FB_ReadXmlLineMsg(
	Prefix:= 'MSG',
	ID:= ,
	File:= 'MSG.xml',
	Text=>);

IF 	Error.Text<>'' THEN
	Error.Text:=CONCAT(Error.Text,sInit.InstName);
	Error.Text:=CONCAT(Error.Text,' :');
	Error.Text:=CONCAT(Error.Text,FB_ReadXmlLineConf.Text);
	Error.Text:=CONCAT(Error.Text,' - ');
	Error.Text:=CONCAT(Error.Text,FB_ReadXmlLineMsg.Text);
END_IF
END_FUNCTION_BLOCK

(* POU zLibrary/Sensopart/FB_Sensopart, ST *)
FUNCTION_BLOCK FB_Sensopart
VAR_INPUT
	b_init							: BOOL;
	b_start							: BOOL;
	b_start_manual					: BOOL;
	b_quitt							: BOOL;
	b_reset							: BOOL;
	b_kamera_aktiv 					: BOOL;
	i16_job							: INT:=1;
	st_Description					: STRING;
END_VAR
VAR_OUTPUT
	b_ready							: BOOL;
	b_done							: BOOL;
	b_busy							: BOOL;
	b_error							: BOOL;

(* Ausgänge der Kamera *)
	Ergebnis_IO						: BOOL;
	Ergebnis_NIO					: BOOL;
	sm_kamera_nicht_bb				: BOOL := FALSE;
	sm_zeitueberschreitung			: BOOL := FALSE;
END_VAR
VAR
	b_first_cycle					: BOOL := TRUE;
	fb_ton_quitt					: TON;
	fb_ton_trigger					: TON;
	fb_tof_trigger					: TOF;
	fb_state_entry					: ST_StateEntry;
	fb_r_trig_start					: R_TRIG;
	fb_r_trig_trigger				: R_TRIG;
END_VAR

VAR_OUTPUT
	(*Sensopart Kamera*)
	a_Trigger 				AT %Q*: BOOL;
	a_Job_Bit1 				AT %Q*: BOOL;
	a_Job_Bit2 				AT %Q*: BOOL;
	a_Job_Bit3 				AT %Q*: BOOL;
	a_Job_Bit4 				AT %Q*: BOOL;
END_VAR
VAR

(* Eingänge von der Kamera *)
	e_Ergebnis_iO			AT %I*: BOOL;
	e_Ergebnis_niO			AT %I*: BOOL;
	e_Betriebsbereit		AT %I*: BOOL;
	e_Best_Jobwechsel		AT %I*: BOOL;
END_VAR
IF b_first_cycle THEN
	b_first_cycle := FALSE;
END_IF

a_Job_Bit1:=i16_job.0;
a_Job_Bit2:=i16_job.1;
a_Job_Bit3:=i16_job.2;
a_Job_Bit4:=i16_job.3;

(* Zeiten *)
fb_ton_quitt(IN:= , PT:= t#100ms, Q=> , ET=> );
fb_ton_trigger(IN:= , PT:= t#150ms, Q=> , ET=> );
fb_tof_trigger(IN:= fb_r_trig_trigger.Q , PT:= t#150ms, Q=> , ET=> );

(* Flanken *)
fb_r_trig_start(CLK:= b_start OR b_start_manual, Q=> );


IF	NOT b_kamera_aktiv THEN
	fb_state_entry.i16_next_step := INAKTIV;
END_IF

(* ==================================Schrittkette================================ *)
fb_state_entry(i16_pos:= 1);

CASE fb_state_entry.i16_step OF
(*=======================================================*)
	INIT_OBJ:
		fb_state_entry.i16_next_step := INIT;

(*=======================================================*)
	INIT:
		IF 	fb_state_entry.E THEN
			b_ready := FALSE;
			b_done := FALSE;
			b_quitt := FALSE;
			b_reset := FALSE;
			b_busy := FALSE;
			b_error := FALSE;
			b_start := FALSE;
			a_Trigger  := FALSE;
			Ergebnis_IO := FALSE;
			Ergebnis_NIO := FALSE;
			sm_kamera_nicht_bb := FALSE;
			sm_zeitueberschreitung := FALSE;
		END_IF

		(*-----------------------Weiterschaltbedingungen----------------------------*)
		IF 	b_init THEN
			IF  NOT b_kamera_aktiv THEN
				fb_state_entry.i16_next_step := BEREIT;		(* Kamera ist inaktiv *)
			ELSE
				fb_state_entry.i16_next_step := 20;			(* Kamera ist aktiv *)
			END_IF
		END_IF

(*=======================================================*)
	20: fb_state_entry.s_debugtext:='Kurze Wartezeit';

		IF 	fb_state_entry.fb_ton_Step.ET > t#300ms THEN
			fb_state_entry.i16_next_step := 30;
		END_IF

(*=======================================================*)
	30: fb_state_entry.s_debugtext:='Kamera Betriebsbereit';

		(*-----------------------Weiterschaltbedingungen----------------------------*)
		IF 	e_Betriebsbereit THEN
			fb_state_entry.i16_next_step := BEREIT;
		ELSIF
		 	fb_state_entry.fb_ton_Step.ET > t#300ms THEN
			sm_kamera_nicht_bb := TRUE;
			fb_state_entry.i16_next_step := FEHLER;
		END_IF

(*=======================================================*)
	BEREIT: fb_state_entry.s_debugtext:='warte auf Start';

		IF fb_state_entry.E THEN
			b_ready := TRUE;
			b_done := TRUE;
		END_IF

		(*-----------------------Weiterschaltbedingungen----------------------------*)
		IF 	b_kamera_aktiv THEN			(* Kamera aktiv *)
			IF 	fb_r_trig_start.Q AND e_Betriebsbereit THEN
				b_start := FALSE;
				b_busy := TRUE;
				b_done := FALSE;
				Ergebnis_IO := FALSE;
				Ergebnis_NIO := FALSE;
				fb_state_entry.i16_next_step := 102;
			ELSIF
				NOT e_Betriebsbereit THEN
				sm_kamera_nicht_bb := TRUE;
				fb_state_entry.i16_next_step := FEHLER;
			END_IF
		ELSE							(* Simulation der Kamera *)
			IF 	fb_r_trig_start.Q THEN
				b_busy := TRUE;
				b_done := FALSE;
				b_start:=FALSE;
				Ergebnis_IO := FALSE;
				Ergebnis_NIO := FALSE;
				fb_state_entry.i16_next_step := 300;
			END_IF
		END_IF

(*=======================================================*)
	102: fb_state_entry.s_debugtext:='Jobwechsel';

		IF 	fb_state_entry.fb_ton_Step.ET > t#1s OR
			e_Best_Jobwechsel THEN
			fb_state_entry.i16_next_step := 105;
		END_IF

(*=======================================================*)
	105: fb_state_entry.s_debugtext:='Kamera wieder bereit';

		IF 	e_Betriebsbereit THEN
			fb_state_entry.i16_next_step := 110;
		ELSIF
			NOT e_Betriebsbereit AND fb_state_entry.fb_ton_Step.ET > t#2s THEN
			sm_kamera_nicht_bb := TRUE;
			fb_state_entry.i16_next_step := FEHLER;
		END_IF

(*=======================================================*)
	110: fb_state_entry.s_debugtext:='Trigger setzen ';

		IF 	fb_state_entry.E THEN
			a_Trigger := TRUE;
			Ergebnis_IO := FALSE;
			Ergebnis_NIO := FALSE;
			fb_ton_trigger.IN := TRUE;
		END_IF

		(*-----------------------Weiterschaltbedingungen----------------------------*)
		IF 	fb_ton_trigger.Q THEN
			a_Trigger := FALSE;
			fb_ton_trigger.IN := FALSE;
			fb_state_entry.i16_next_step := 130;
		END_IF

(*=======================================================*)
	120: fb_state_entry.s_debugtext:='Warten auf Ergebnis der Kamera';

		IF 	NOT e_Ergebnis_iO AND
			NOT e_Ergebnis_niO THEN
			fb_state_entry.i16_next_step := 130;
		ELSIF
			fb_state_entry.fb_ton_Step.ET > t#4000ms THEN
			sm_zeitueberschreitung := TRUE;
			fb_state_entry.i16_next_step := FEHLER;
		END_IF

(*=======================================================*)
	130: fb_state_entry.s_debugtext:='Warten auf Ergebnis der Kamera ';

		IF 	NOT fb_state_entry.E AND e_Ergebnis_iO AND e_Betriebsbereit THEN
			Ergebnis_IO := TRUE;
			fb_state_entry.i16_next_step := BEREIT;
		ELSIF
			NOT fb_state_entry.E AND e_Ergebnis_niO AND e_Betriebsbereit THEN
			Ergebnis_NIO := TRUE;
			fb_state_entry.i16_next_step := BEREIT;
		ELSIF
			fb_state_entry.fb_ton_Step.ET > t#4000ms THEN
			sm_zeitueberschreitung := TRUE;
			fb_state_entry.i16_next_step := FEHLER;
		END_IF

		IF 	fb_state_entry.X THEN
			b_busy := FALSE;
			b_done := TRUE;
		END_IF

(*=======================================================*)
	300: fb_state_entry.s_debugtext:='Kamera ist nicht aktiv (Warten) ';		

		IF 	fb_state_entry.fb_ton_Step.ET > t#500ms THEN
			b_busy := FALSE;
			b_done := TRUE;
			Ergebnis_IO := TRUE;
			fb_state_entry.i16_next_step := BEREIT;
		END_IF

(*=======================================================*)
	STOP, FEHLER:
		IF 	fb_state_entry.E THEN
			b_error := TRUE;
			fb_ton_quitt.IN := FALSE;
			a_Trigger := FALSE;
		END_IF

		(*-----------------------Weiterschaltbedingungen----------------------------*)
		IF	(b_reset OR b_quitt) AND
			NOT fb_state_entry.E THEN
			b_error := FALSE;
			fb_ton_quitt.IN := TRUE;
		END_IF

		IF 	fb_ton_quitt.Q THEN
			fb_ton_quitt.IN := FALSE;
			fb_state_entry.i16_next_step := INIT;
		END_IF

(*=======================================================*)
	INAKTIV:
		IF 	fb_state_entry.E THEN
			b_ready := FALSE;
			b_done := FALSE;
			b_busy := FALSE;
			b_start := FALSE;
		END_IF

		IF	b_kamera_aktiv THEN
			fb_state_entry.i16_next_step := STOP;
		END_IF

END_CASE

fb_state_entry(i16_pos:= 2);
END_FUNCTION_BLOCK

(* POU zLibrary/Sensopart/FB_SensopartEthernet, ST *)
FUNCTION_BLOCK FB_SensopartEthernet
VAR_INPUT
	Activated				: BOOL;
	JobNo					: INT;
	s_IpAdress				: STRING;
	i_DataPort				: UDINT;
	i_CmdPort				: UDINT;
	st_ctrl_in				: struct_ctrl_in;
	st_Description			: STRING;
	st_InstName				: STRING;
	SensopartErgebnis		: STRING(15); (*Ergebnis Sensopart Kamera*)
END_VAR
VAR_IN_OUT

END_VAR
VAR_OUTPUT
	st_ctrl_out				: struct_ctrl_out;
	Connected				: BOOL;							(* Sockets Connected*)
	RecvDataString			: T_MaxString;
	ActJobNo				: INT;
END_VAR
VAR
	fb_ton_quitt						: TON;
	fb_state_entry					: ST_StateEntry;
	fb_state_entry_command			: ST_StateEntry;

	(* Error Handling *)
	FB_ReadXmlLineConf			: FB_ReadXmlLine;
	FB_ReadXmlLineMsg			: FB_ReadXmlLine;
	(*Variablen für Behr Meldungen*)
	TempErrorText					: STRING(255);
	ProcessTime					: DINT;				(* Counts the time in steps of 100ms since starting operation *)
	Error							: ErrorStruct;

	sm_kamera_keine_reaktion		: BOOL;
	sm_kamera_nicht_bb			: BOOL;
	sm_jobnummer_nicht_erlaubt		: BOOL;		(* erlaubter Bereich von 1-255 *)
	sm_kamera_command_error		: BOOL;
	sm_kamera_connect_error		: BOOL;
	sm_kamera_send_error			: BOOL;
	sm_kamera_rec_error			: BOOL;

	(*TcpIp-Connection via Socket*)
	FBClientServerConnectionCmd 	: FB_ClientServerConnection;
	FBClientServerConnectionRcv 	: FB_ClientServerConnection;
	FBSocketSend					: FB_SocketSend;
	FBSocketRecv					: FB_SocketReceive;
	SocketHandleCmd				: T_HSOCKET;
	SocketHandleRcv				: T_HSOCKET;
	ErrorId						: UDINT;
	nRecBytes					: UDINT;						(* Contains the number of bytes currently received. *)

	RecvStringCmd				: STRING(25);

	TRG_CMD:		ARRAY [0..2] OF BYTE:= 16#54,16#52,16#47;	(* [T, R, G] Trigger *)
	CJB_CMD:		ARRAY [0..5] OF BYTE:= 16#43,16#4A,16#42;	(* [C, J, B, 0, 0, 1] ChangeJoB z.B für Jobnummer 1 *)
	CJB_RCV:		ARRAY [0..7] OF BYTE;

	JbNoMem					: INT;
	CalcJbNo					: BYTE;

	b_Kam_Pruef_IO			:BOOL; 				(* Kameraprüfung Ergebnis iO *)
	b_Kam_Pruef_NIO			:BOOL; 				(* Kameraprüfung Ergebnis niO *)

	b_Kam_Bereit	  			: BOOL;				(* Bereit für nächsten ext. Trigger *)
	b_Betriebsbereit_eth			: BOOL:=FALSE;	(* Bereit kommt von EtherNet (noch nicht programmiert) *)
	e_Betriebsbereit  		AT %I*: BOOL;			(* Bereit kommt nur über Hardware-Eingang *)
 	BtnConnect					: sButtonVisu;
	BtnTrigger					: sButtonVisu;

END_VAR
(* Zeiten *)
fb_ton_quitt(IN:= , PT:= t#100ms, Q=> , ET=> );

(* Aufrufe *)
Btn_Init();
Command();
ErrorHandling();

b_Kam_Bereit := e_Betriebsbereit OR b_Betriebsbereit_eth;	(* Betriebsbereit  von EtherNet oder Eingang *)

(* Toplevel *)
IF	NOT Activated THEN
	fb_state_entry.i16_next_step := INAKTIV;
END_IF

IF fb_state_entry.i16_next_step > INIT AND fb_state_entry.i16_next_step < FEHLER THEN
	IF fb_state_entry.i16_next_step < STOP THEN
		IF st_ctrl_in.b_stop THEN
			fb_state_entry.i16_next_step := STOP;
		END_IF
		IF 	sm_kamera_command_error OR
			sm_kamera_send_error OR
			sm_kamera_rec_error OR
			sm_kamera_connect_error THEN
			fb_state_entry.i16_next_step := FEHLER;
		END_IF
	END_IF
END_IF

(* ==================================Schrittkette================================ *)
fb_state_entry(i16_pos:= 1);

CASE fb_state_entry.i16_step OF
(*=======================================================*)
INIT_OBJ:

	fb_state_entry.i16_next_step := INIT;

(*=======================================================*)
INIT:
	IF 	fb_state_entry.E THEN
		fb_ton_quitt.IN := FALSE;
		st_ctrl_out := st_ctrl_out_Empty;
		b_Kam_Pruef_IO := FALSE;
		b_Kam_Pruef_NIO := FALSE;
		sm_kamera_nicht_bb := FALSE;
		sm_kamera_keine_reaktion := FALSE;
		sm_jobnummer_nicht_erlaubt := FALSE;
		sm_kamera_command_error:=FALSE;
		sm_kamera_connect_error:=FALSE;
		sm_kamera_send_error:=FALSE;
		sm_kamera_rec_error:=FALSE;
		Error.No:=0;
		Error.Text:='';
	END_IF

	(*-----------------------Weiterschaltbedingungen----------------------------*)
	IF	BtnConnect.tasten OR
		st_ctrl_in.b_init THEN
		fb_state_entry.i16_next_step := 30;
	END_IF

(*=======================================================*)
30: fb_state_entry.s_debugtext:='start Connect';

	IF	fb_state_entry.E THEN
		fb_state_entry_command.i16_next_step:=20;
	END_IF

	(*-----------------------Weiterschaltbedingungen----------------------------*)
	IF 	fb_state_entry_command.i16_step > INIT THEN
		fb_state_entry.i16_next_step := 35;
	ELSIF
		fb_state_entry.fb_ton_Step.ET > t#2s THEN
		sm_kamera_nicht_bb := TRUE;
		fb_state_entry.i16_next_step := FEHLER;
	END_IF

(*=======================================================*)
35: fb_state_entry.s_debugtext:='warte auf bereit von connect';

	IF 	fb_state_entry_command.i16_step = BEREIT THEN
		fb_state_entry.i16_next_step := BEREIT;
	ELSIF
		fb_state_entry.fb_ton_Step.ET > t#20s THEN
		sm_kamera_nicht_bb := TRUE;
		fb_state_entry.i16_next_step := FEHLER;
	END_IF

(*=======================================================*)
BEREIT: fb_state_entry.s_debugtext:='warte auf Start';

	IF 	fb_state_entry.E THEN
		st_ctrl_out.b_bereit := TRUE;
		st_ctrl_in.b_start:=FALSE;
	END_IF

	(*-----------------------Weiterschaltbedingungen----------------------------*)
	IF 	(b_Kam_Bereit OR NOT Activated) AND
		(st_ctrl_in.b_start OR BtnTrigger.tasten) THEN
		b_Kam_Pruef_IO := FALSE;
		b_Kam_Pruef_NIO := FALSE;
		fb_state_entry.i16_next_step := 110;
	ELSIF
		fb_state_entry.fb_ton_Step.ET > t#1s AND
		(NOT b_Kam_Bereit OR NOT Connected) AND
		Activated THEN
		sm_kamera_nicht_bb := TRUE;
		fb_state_entry.i16_next_step := FEHLER;
	END_IF

	IF 	fb_state_entry.X THEN
		st_ctrl_out.b_busy:=TRUE;
		st_ctrl_out.b_bereit := FALSE;
		st_ctrl_out.b_fertig := FALSE;
	END_IF

(*=======================================================*)
110: fb_state_entry.s_debugtext:='Jobnummer im erlaubten Bereich?';

	(*-----------------------Weiterschaltbedingungen----------------------------*)
	IF 	JobNo > 0 AND
		JobNo < 256 THEN
		fb_state_entry.i16_next_step := 120;
	ELSE
		sm_jobnummer_nicht_erlaubt := TRUE;
		fb_state_entry.i16_next_step := FEHLER;
	END_IF

(*=======================================================*)
120: fb_state_entry.s_debugtext:='Trigger setzen';

	IF 	fb_state_entry.E THEN
		fb_state_entry_command.i16_next_step:=110;
		b_Kam_Pruef_IO := FALSE;
		b_Kam_Pruef_NIO := FALSE;
	END_IF

	(*-----------------------Weiterschaltbedingungen----------------------------*)
	IF 	fb_state_entry_command.i16_step > BEREIT THEN
		fb_state_entry.i16_next_step := 130;
	ELSIF
		fb_state_entry.fb_ton_Step.ET > t#3s THEN
		sm_kamera_keine_reaktion := TRUE;
		fb_state_entry.i16_next_step := FEHLER;
	END_IF

(*=======================================================*)
130: fb_state_entry.s_debugtext:='warte bis Kamera fertig ist';

	(*-----------------------Weiterschaltbedingungen----------------------------*)
	IF 	fb_state_entry_command.i16_step = BEREIT THEN
		fb_state_entry.i16_next_step := 140;
	ELSIF
		fb_state_entry.fb_ton_Step.ET > t#5s THEN
		sm_kamera_keine_reaktion := TRUE;
		fb_state_entry.i16_next_step := FEHLER;
	END_IF

(*=======================================================*)
140: fb_state_entry.s_debugtext:='Ergebnis der Kamera auswerten';

	(*-----------------------Weiterschaltbedingungen----------------------------*)
	(*// RecvDataString Erklärung
	// 2 = Anzahl der Ausgangsbits der Kamera
	// P = Positives Ergebnis
	// F = Negatives Ergebnis
	// Jobnummer
	// evtl. Jobnummer anders abfragen*)
	IF 	RecvDataString = CONCAT(SensopartErgebnis, INT_TO_STRING(JobNo)) THEN		(* Stecker iO *)
		b_Kam_Pruef_IO :=  TRUE;
		fb_state_entry.i16_next_step := BEREIT;
	ELSE		(* Stecker niO *)
		b_Kam_Pruef_NIO :=  TRUE;
		fb_state_entry.i16_next_step := BEREIT;
	END_IF

	IF 	fb_state_entry.X THEN
		st_ctrl_out.b_busy:=FALSE;
		st_ctrl_out.b_fertig := TRUE;
	END_IF

(*=======================================================*)
STOP, FEHLER:

	IF 	fb_state_entry.E THEN
		st_ctrl_out := st_ctrl_out_Empty;
		st_ctrl_out.b_gestoppt := fb_state_entry.i16_next_step = STOP;
		st_ctrl_out.b_fehler := fb_state_entry.i16_next_step = FEHLER;
		fb_state_entry_command.i16_next_step:= fb_state_entry.i16_next_step;
		fb_ton_quitt.IN := FALSE;
	END_IF

	IF	sm_kamera_keine_reaktion THEN
		FB_ReadXmlLineMsg.ID:='sm_kamera_keine_reaktion';
		Error.No:=1;
	ELSIF
		sm_kamera_nicht_bb THEN
		FB_ReadXmlLineMsg.ID:='sm_kamera_nicht_bb';
		Error.No:=2;
	ELSIF
		sm_jobnummer_nicht_erlaubt THEN
		FB_ReadXmlLineMsg.ID:='sm_jobnummer_nicht_erlaubt';
		Error.No:=3;
	ELSIF
		sm_kamera_command_error THEN
		FB_ReadXmlLineMsg.ID:='sm_kamera_command_error';
		Error.No:=4;
	ELSIF
		sm_kamera_connect_error THEN
		FB_ReadXmlLineMsg.ID:='sm_kamera_connect_error';
		Error.No:=5;
	ELSIF
		sm_kamera_send_error THEN
		FB_ReadXmlLineMsg.ID:='sm_kamera_send_error';
		Error.No:=6;
	ELSIF
		sm_kamera_rec_error THEN
		FB_ReadXmlLineMsg.ID:='sm_kamera_rec_error';
		Error.No:=7;
	END_IF

	(*-----------------------Weiterschaltbedingungen----------------------------*)
	IF 	(st_ctrl_in.b_quitt OR gResetAll) THEN
		fb_ton_quitt.IN := TRUE;
	END_IF

	IF 	fb_ton_quitt.Q THEN
		fb_ton_quitt.IN := FALSE;
		fb_state_entry.i16_next_step := INIT;
	END_IF

(*=======================================================*)
INAKTIV:

	IF 	fb_state_entry.E THEN
		st_ctrl_out := st_ctrl_out_Empty;
	END_IF

	st_ctrl_out.b_bereit := TRUE;
	IF	Activated THEN
		fb_state_entry.i16_next_step := INIT;
	END_IF

END_CASE

fb_state_entry(i16_pos:= 2);
st_ctrl_in := st_ctrl_in_Empty;
END_FUNCTION_BLOCK
ACTION Btn_Init:
(*=====================================================================*)
BtnConnect.Text:='Connect';
BtnConnect.BackgroundColor:=Color.darkgrey;
BtnConnect.Enable:= TRUE; (*ModeSelect.Mode <> MODE_MANUAL;*)
IF	BtnConnect.Enable THEN
	BtnConnect.TextColor:=Color.grey;
ELSE
	BtnConnect.TextColor:=Color.black;
END_IF
BtnConnect.Visible:=TRUE;

(*=====================================================================*)
BtnTrigger.Text:='Trigger';
BtnTrigger.BackgroundColor:=Color.darkgrey;
BtnTrigger.Enable:= TRUE; (* ModeSelect.Mode <> MODE_MANUAL;*)
IF	BtnTrigger.Enable THEN
	BtnTrigger.TextColor:=Color.grey;
ELSE
	BtnTrigger.TextColor:=Color.black;
END_IF
BtnTrigger.Visible:=TRUE;
END_ACTION
ACTION Command:
(*TemplateClass01_Function01: write here a short Description of this command*)

Connected:=	FBClientServerConnectionCmd.eState=eSOCKET_CONNECTED AND
				FBClientServerConnectionRcv.eState=eSOCKET_CONNECTED;

(* ==================================Schrittkette================================ *)
fb_state_entry_command(i16_pos:= 1);

CASE fb_state_entry_command.i16_step OF

INIT_OBJ:

	fb_state_entry_command.i16_next_step:=INIT;

(*===========================================================*)
INIT: fb_state_entry_command.s_debugtext:= 'INIT kommt vom Hauptablauf';

(*===========================================================*)
20:	fb_state_entry_command.s_debugtext:='Preset local Vars';

	FBClientServerConnectionCmd(bEnable:=FALSE);
	FBClientServerConnectionRcv(bEnable:=FALSE);
	FBSocketSend(bExecute:=FALSE);
	FBSocketRecv(bExecute:=FALSE);
	fb_state_entry_command.i16_next_step:=30;

(*===========================================================*)
30:	fb_state_entry_command.s_debugtext:='Create new Socket-Connection: Start';

	FBClientServerConnectionCmd
		(bEnable		:=TRUE,
		nMode			:=CONNECT_MODE_ENABLEDBG,	(* Enable Debugging (to see in SystemManager Logger*)
		sRemoteHost	:=s_IpAdress,						(* IP-Adresse NewPort-Achsregler *)
		nRemotePort	:=i_CmdPort,						(* TCPIP Socket Port *)
		tReconnect		:= t#10s);
	IF 	FBClientServerConnectionCmd.bBusy THEN
		fb_state_entry_command.i16_next_step:=40;
	END_IF

(*===========================================================*)
40:	fb_state_entry_command.s_debugtext:='Create new Socket-Connection: Finished';

	FBClientServerConnectionCmd
		(bEnable		:=TRUE,
		nMode			:=CONNECT_MODE_ENABLEDBG,	(* Enable Debugging (to see in SystemManager Logger*)
		sRemoteHost	:=s_IpAdress,						(* IP-Adresse NewPort-Achsregler *)
		nRemotePort	:=i_CmdPort,						(* TCPIP Socket Port *)
		tReconnect		:= t#10s);
	IF 	NOT FBClientServerConnectionCmd.bBusy AND
		NOT FBClientServerConnectionCmd.bError THEN
		SocketHandleCmd:=FBClientServerConnectionCmd.hSocket;
		fb_state_entry_command.i16_next_step:=50;
	ELSIF
		FBClientServerConnectionCmd.bError THEN
		sm_kamera_connect_error:=TRUE;
		fb_state_entry_command.i16_next_step:=FEHLER;
		ErrorId:=FBClientServerConnectionCmd.nErrId;
	END_IF

(*===========================================================*)
50:	fb_state_entry_command.s_debugtext:='Create new Socket-Connection: Start';

	FBClientServerConnectionRcv
		(bEnable		:=TRUE,
		nMode			:=CONNECT_MODE_ENABLEDBG,	(* Enable Debugging (to see in SystemManager Logger*)
		sRemoteHost	:=s_IpAdress,						(* IP-Adresse NewPort-Achsregler *)
		nRemotePort	:=i_DataPort,						(* TCPIP Socket Port *)
		tReconnect		:= t#10s);
	IF 	FBClientServerConnectionRcv.bBusy THEN
		fb_state_entry_command.i16_next_step:=60;
	END_IF

(*===========================================================*)
60:	fb_state_entry_command.s_debugtext:='Create new Socket-Connection: Finished';

	FBClientServerConnectionRcv
		(bEnable		:=TRUE,
		nMode			:=CONNECT_MODE_ENABLEDBG,	(* Enable Debugging (to see in SystemManager Logger*)
		sRemoteHost	:=s_IpAdress,						(* IP-Adresse NewPort-Achsregler *)
		nRemotePort	:=i_DataPort,						(* TCPIP Socket Port *)
		tReconnect		:= t#10s);
	IF 	NOT FBClientServerConnectionRcv.bBusy AND
		NOT FBClientServerConnectionRcv.bError THEN
		SocketHandleRcv:=FBClientServerConnectionRcv.hSocket;
		fb_state_entry_command.i16_next_step:=70;
	ELSIF
		FBClientServerConnectionRcv.bError THEN
		sm_kamera_connect_error:=TRUE;
		fb_state_entry_command.i16_next_step:=FEHLER;
		ErrorId:=FBClientServerConnectionRcv.nErrId;
	END_IF

(*===========================================================*)
70:	fb_state_entry_command.s_debugtext:='Check if Socket is correct connected';

	IF 	Connected AND
		SocketHandleCmd.handle>0 AND
		SocketHandleRcv.handle>0 THEN
		fb_state_entry_command.i16_next_step:=BEREIT;
	END_IF

(*=======================================================*)
BEREIT: fb_state_entry_command.s_debugtext:= 'START kommt vom Hauptablauf';

(*===========================================================*)
110: fb_state_entry_command.s_debugtext:='Check if Socket is correct connected';

	IF 	Connected AND
		SocketHandleCmd.handle>0 AND
		SocketHandleRcv.handle>0 AND
		b_Kam_Bereit AND
		Activated THEN
		IF 	JobNo=0 THEN
		 	 fb_state_entry_command.i16_next_step:=FEHLER;
		ELSE
			MEMSET(destAddr:=ADR(RecvDataString), fillByte:=0, n:=SIZEOF(RecvDataString));
			MEMSET(destAddr:=ADR(CJB_RCV), fillByte:=0, n:=SIZEOF(CJB_RCV));
			MEMSET(destAddr:=ADR(RecvStringCmd), fillByte:=0, n:=SIZEOF(RecvStringCmd));
			fb_state_entry_command.i16_next_step:=120;
		END_IF
	ELSE
		sm_kamera_connect_error:=TRUE;
		fb_state_entry_command.i16_next_step:=FEHLER;
	END_IF

(*===========================================================*)
120: fb_state_entry_command.s_debugtext:='Job-Nummer prüfen und setzen.';

	 IF 	JobNo <> ActJobNo THEN
		JbNoMem:=JobNo;
		CalcJbNo:=INT_TO_BYTE(JbNoMem/100);
		CJB_CMD[3]:=16#30+CalcJbNo;

		CalcJbNo:=CalcJbNo*100;
		JbNoMem:=JbNoMem-CalcJbNo;
		CalcJbNo:=INT_TO_BYTE(JbNoMem/10);
		CJB_CMD[4]:=16#30+CalcJbNo;

		CalcJbNo:=CalcJbNo*10;
		JbNoMem:=INT_TO_BYTE(JbNoMem-CalcJbNo);
		CJB_CMD[5]:=16#30+INT_TO_BYTE(JbNoMem);

		fb_state_entry_command.i16_next_step:=130;
	ELSE
		fb_state_entry_command.i16_next_step:=200;
	END_IF

(*===========================================================*)
130: fb_state_entry_command.s_debugtext:='start FBSocketSend';

	FBSocketSend(bExecute	:=TRUE,
				hSocket		:= SocketHandleCmd,
				cbLen			:= 6,
				pSrc			:= ADR(CJB_CMD),
				tTimeout		:= t#5s);
	IF 	FBSocketSend.bBusy THEN
		fb_state_entry_command.i16_next_step:=140;
	END_IF

(*===========================================================*)
140: fb_state_entry_command.s_debugtext:='warte auf fertig  FBSocketSend';

	FBSocketSend(bExecute:=FALSE);
	IF 	NOT FBSocketSend.bBusy AND
		NOT FBSocketSend.bError THEN
		fb_state_entry_command.i16_next_step:=150;
	ELSIF
		FBSocketSend.bError THEN
		sm_kamera_send_error:=TRUE;
		fb_state_entry_command.i16_next_step:=FEHLER;
		ErrorId:=FBSocketSend.nErrId;
	END_IF

(*===========================================================*)
150: fb_state_entry_command.s_debugtext:='Wait before Receive';

	IF 	fb_state_entry_command.fb_ton_Step.ET > T#0ms THEN
		fb_state_entry_command.i16_next_step:=160;
	END_IF

(*===========================================================*)
160: fb_state_entry_command.s_debugtext:='Receive starten';

	FBSocketRecv(	bExecute	:=TRUE,
					hSocket	:= SocketHandleCmd,
					cbLen		:= SIZEOF(CJB_RCV),
					pDest		:= ADR(CJB_RCV),
					tTimeout	:= t#5s );
	IF 	FBSocketRecv.bBusy THEN
		fb_state_entry_command.i16_next_step:=170;
	END_IF

(*===========================================================*)
170: fb_state_entry_command.s_debugtext:='Job-Nr. rücklesen';

	FBSocketRecv(bExecute:=FALSE);
	IF 	NOT FBSocketRecv.bBusy AND
		NOT FBSocketRecv.bError THEN
		nRecBytes:=FBSocketRecv.nRecBytes;
		fb_state_entry_command.i16_next_step:=180;
	ELSIF
		FBSocketRecv.bError THEN
		sm_kamera_rec_error:=TRUE;
		fb_state_entry_command.i16_next_step:=FEHLER;
		ErrorId:=FBSocketRecv.nErrId;
	END_IF

(*===========================================================*)
180: fb_state_entry_command.s_debugtext:='Empfangene Daten gültig';

	IF 	nRecBytes>0 THEN
		fb_state_entry_command.i16_next_step:=190;
	ELSE
		fb_state_entry_command.i16_next_step:=160;
	END_IF

(*===========================================================*)
190: fb_state_entry_command.s_debugtext:='prüfe Ergebniss';

	IF 	CJB_RCV[3] < 16#50 THEN
		ErrorId:=16#0040;
		sm_kamera_rec_error:=TRUE;
		fb_state_entry_command.i16_next_step:=FEHLER;
	ELSIF
		CJB_RCV[5] <> CJB_CMD[3] OR
		CJB_RCV[6] <> CJB_CMD[4] OR
		CJB_RCV[7] <> CJB_CMD[5] THEN
		ErrorId:=16#0050;
		sm_kamera_rec_error:=TRUE;
		fb_state_entry_command.i16_next_step:=FEHLER;
	ELSE
		ErrorId:=16#0000;
		ActJobNo:=(CJB_RCV[5]-16#30)*100+(CJB_RCV[6]-16#30)*10+(CJB_RCV[7]-16#30);
	 	fb_state_entry_command.i16_next_step:=200;
	END_IF

(*===========================================================*)
(*===========================================================*)
200: fb_state_entry_command.s_debugtext:='Trigger-Cmd senden';

	FBSocketSend(bExecute	:=TRUE,
				hSocket		:= SocketHandleCmd,
				cbLen			:= 3,
				pSrc			:= ADR(TRG_CMD),
				tTimeout		:= T#5S);
	IF 	FBSocketSend.bBusy THEN
		fb_state_entry_command.i16_next_step:=210;
	END_IF

(*===========================================================*)
210: fb_state_entry_command.s_debugtext:='warte auf fertig Trigger-Cmd';

	FBSocketSend(bExecute:=FALSE);
	IF 	NOT FBSocketSend.bBusy AND
		NOT FBSocketSend.bError THEN
		fb_state_entry_command.i16_next_step:=220;
	ELSIF
		FBSocketSend.bError THEN
		sm_kamera_send_error:=TRUE;
		fb_state_entry_command.i16_next_step:=FEHLER;
		ErrorId:=FBSocketSend.nErrId;
	END_IF

(*===========================================================*)
220: fb_state_entry_command.s_debugtext:='Wait before Receive';

	IF 	fb_state_entry_command.fb_ton_Step.ET > t#10ms THEN
		fb_state_entry_command.i16_next_step:=230;
	END_IF

(*===========================================================*)
230: fb_state_entry_command.s_debugtext:='Receive starten';

	FBSocketRecv(	bExecute	:=TRUE,
					hSocket	:= SocketHandleCmd,
					cbLen		:= SIZEOF(RecvStringCmd),
					pDest		:= ADR(RecvStringCmd),
					tTimeout	:= t#5s );
	IF 	FBSocketRecv.bBusy THEN
		fb_state_entry_command.i16_next_step:=240;
	END_IF

(*===========================================================*)
240: fb_state_entry_command.s_debugtext:='Receive-Buffer lesen';

	FBSocketRecv(bExecute:=FALSE);
	IF 	NOT FBSocketRecv.bBusy AND
		NOT FBSocketRecv.bError THEN
		nRecBytes:=FBSocketRecv.nRecBytes;
		fb_state_entry_command.i16_next_step:=250;
	ELSIF
		FBSocketRecv.bError THEN
		sm_kamera_rec_error:=TRUE;
		fb_state_entry_command.i16_next_step:=FEHLER;
		ErrorId:=FBSocketRecv.nErrId;
	END_IF

(*===========================================================*)
250: fb_state_entry_command.s_debugtext:='Response erhalten?';

	IF 	nRecBytes>0 THEN
		fb_state_entry_command.i16_next_step:=300;
	ELSE
		fb_state_entry_command.i16_next_step:=230;		(*wdh. bis etwas ankommt*)
	END_IF

(*===========================================================*)
(*===========================================================*)
300: fb_state_entry_command.s_debugtext:='Ergebnis-Daten von Datenport lesen';

	IF 	Activated THEN
		fb_state_entry_command.i16_next_step:=310;
	ELSE
		fb_state_entry_command.i16_next_step:=BEREIT;
	END_IF

(*===========================================================*)
310: fb_state_entry_command.s_debugtext:='Receive starten';

	FBSocketRecv(bExecute	:=TRUE,
				hSocket		:= SocketHandleRcv,
				cbLen			:= SIZEOF(RecvDataString),
				pDest			:= ADR(RecvDataString),
				tTimeout		:= T#5S );
	IF 	FBSocketRecv.bBusy THEN
		fb_state_entry_command.i16_next_step:=320;
	END_IF

(*===========================================================*)
320: fb_state_entry_command.s_debugtext:='Receive-Buffer lesen';

	FBSocketRecv(bExecute:=FALSE);
	IF 	NOT FBSocketRecv.bBusy AND
		NOT FBSocketRecv.bError THEN
		nRecBytes:=FBSocketRecv.nRecBytes;
		fb_state_entry_command.i16_next_step:=330;
	ELSIF
		FBSocketRecv.bError THEN
		sm_kamera_rec_error:=TRUE;
		fb_state_entry_command.i16_next_step:=FEHLER;
		ErrorId:=FBSocketRecv.nErrId;
	END_IF

(*===========================================================*)
330: fb_state_entry_command.s_debugtext:='Antwort erhalten?';

	IF 	nRecBytes>0 THEN
		fb_state_entry_command.i16_next_step:=BEREIT;
	ELSE
		fb_state_entry_command.i16_next_step:=310;		(*wdh. bis etwas ankommt*)
	END_IF

(*=======================================================*)
STOP, FEHLER:

	IF 	fb_ton_quitt.Q THEN
		fb_state_entry_command.i16_next_step := INIT;
	END_IF

END_CASE

fb_state_entry_command(i16_pos:= 2);
END_ACTION
ACTION ErrorHandling:
(*------------------------------------------------------------------
	Error-Handling
  ------------------------------------------------------------------*)

FB_ReadXmlLineConf(
	Prefix:= 'CONFIG',
	ID:= st_InstName,
	File:= 'CONFIG.xml',
	Text=>  );

FB_ReadXmlLineMsg(
	Prefix:= 'MSG',
	ID:= ,
	File:= 'MSG.xml',
	Text=>);

IF	NOT st_ctrl_out.b_fehler THEN	(*OR NOT Activated *)
	Error.No:=0;
	Error.Text:='';
	TempErrorText:='';
END_IF

IF 	Error.Text<>''	AND ST_Lng.b_EndChangeLng THEN
	Error.Typ:=0;
	ErrorHandler.AddError(ErrorToAdd:=Error,
						sVisu:=Visu.ErrorHandler);
END_IF

IF	 st_ctrl_out.b_fehler THEN
	Error.Text:=FB_ReadXmlLineConf.Text;
	Error.Text:=CONCAT(Error.Text,': ');
	Error.Text:=CONCAT(Error.Text,FB_ReadXmlLineMsg.Text);
END_IF
END_ACTION

(* Visualisation zLibrary/ept/DataBehr/Data_BOOL
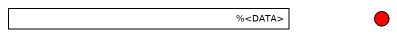
rectangle at (0,0)-(281,21): text "%<DATA>"; shows $Beschreibung$; invisible if $unsichtbar$
ellipse at (366,3)-(381,18): invisible if $unsichtbar$; alarm colour if $value$
2 elements of other kinds (tables, trends, ...) not read
*)

(* Visualisation zLibrary/ept/DataBehr/DATA_DEZIMAL
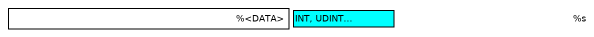
rectangle at (0,0)-(281,21): text "%<DATA>"; shows $Beschreibung$; invisible if $unsichtbar$; tooltip $Beschreibung$
rectangle at (560,0)-(761,21): text "%s"; shows '$Einheit$'; invisible if $unsichtbar$; tooltip $Einheit$
rectangle at (285,2)-(386,19): text "INT, UDINT..."; invisible if TRUE
2 elements of other kinds (tables, trends, ...) not read
*)

(* Visualisation zLibrary/ept/DataBehr/DATA_DEZIMAL_REAL
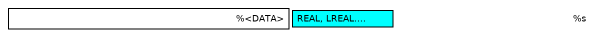
rectangle at (0,0)-(281,21): text "%<DATA>"; shows $Beschreibung$; invisible if $unsichtbar$; tooltip $Beschreibung$
rectangle at (560,0)-(761,21): text "%s"; shows '$Einheit$'; invisible if $unsichtbar$; tooltip $Einheit$
rectangle at (284,2)-(385,19): text "REAL, LREAL...."; invisible if TRUE
2 elements of other kinds (tables, trends, ...) not read
*)

(* Visualisation zLibrary/ept/Data/DATA_HEADER
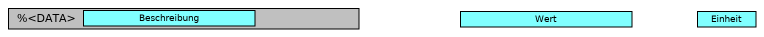
rectangle at (0,0)-(351,21): text "%<DATA>"; shows 'Description'
rectangle at (75,2)-(247,18): text "Beschreibung"; invisible if TRUE
rectangle at (452,3)-(624,19): text "Wert"; invisible if TRUE
rectangle at (689,3)-(748,19): text "Einheit"; invisible if TRUE
2 elements of other kinds (tables, trends, ...) not read
*)

(* Visualisation zLibrary/ept/DataBehr/DATA_HEADER_BEER
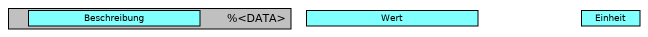
rectangle at (0,0)-(283,21): text "%<DATA>"; shows 'Description'
rectangle at (20,2)-(192,18): text "Beschreibung"; invisible if TRUE
rectangle at (298,2)-(470,18): text "Wert"; invisible if TRUE
rectangle at (573,2)-(632,18): text "Einheit"; invisible if TRUE
2 elements of other kinds (tables, trends, ...) not read
*)

(* Visualisation zLibrary/ept/Data/DATA_LINE
2 elements of other kinds (tables, trends, ...) not read
*)

(* Visualisation zLibrary/ept/Data/DATA_LINE_B
3 elements of other kinds (tables, trends, ...) not read
*)

(* Visualisation zLibrary/ept/Data/DATA_LINE_BYTE
4 elements of other kinds (tables, trends, ...) not read
*)

(* Visualisation zLibrary/ept/Data/DATA_LINE_I16
4 elements of other kinds (tables, trends, ...) not read
*)

(* Visualisation zLibrary/ept/Data/Data_LINE_i32
4 elements of other kinds (tables, trends, ...) not read
*)

(* Visualisation zLibrary/ept/Data/DATA_LINE_LR
4 elements of other kinds (tables, trends, ...) not read
*)

(* Visualisation zLibrary/ept/Data/DATA_LINE_STR
3 elements of other kinds (tables, trends, ...) not read
*)

(* Visualisation zLibrary/ept/DataBehr/DATA_STRING
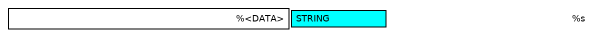
rectangle at (0,0)-(281,21): text "%<DATA>"; shows $Beschreibung$; invisible if $unsichtbar$
rectangle at (562,0)-(763,21): text "%s"; shows '$Einheit$'; invisible if $unsichtbar$; tooltip $Einheit$
rectangle at (283,2)-(378,19): text "STRING"; invisible if TRUE
2 elements of other kinds (tables, trends, ...) not read
*)

(* Visualisation 02_TypeData/DIALOG_SAVE_AS
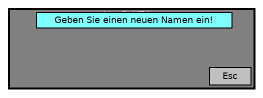
rectangle at (1,0)-(248,81): text "%<DATA>"; shows 'save_as'
rectangle at (29,4)-(225,20): text "Geben Sie einen neuen Namen ein!"; invisible if TRUE
rectangle at (202,59)-(244,77): text "Esc"; toggles TDHandler.b_Dialog_save_as_on
1 elements of other kinds (tables, trends, ...) not read
*)

(* Visualisation zLibrary/ept/Dig_IN_OUT/DIGIN
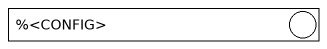
rounded rectangle at (1,1)-(280,32): text "%<CONFIG>"; shows '$Input$'
ellipse at (281,3)-(308,30): alarm colour if $Station$.$Input$; tooltip $Input$
1 more shapes without text or variables
*)

(* Visualisation zLibrary/ept/Dig_IN_OUT/DIGIN_red
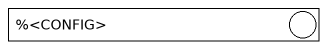
rounded rectangle at (1,1)-(280,32): text "%<CONFIG>"; shows '$Input$'
ellipse at (281,3)-(308,30): alarm colour if $Station$.$Input$; tooltip $Input$
1 more shapes without text or variables
*)

(* Visualisation zLibrary/ept/Dig_IN_OUT/DIGOUT_SMAL
4 elements of other kinds (tables, trends, ...) not read
*)

(* Visualisation zLibrary/ept/Dig_IN_OUT/DIGOUT_TOUCH_SMAL
rectangle at (0,0)-(311,33): taps $Station$.$Output$
4 elements of other kinds (tables, trends, ...) not read
*)

(* Visualisation zLibrary/ept/DOOR_LOCK
rectangle at (0,0)-(31,31): invisible if $lock$ AND NOT $visibal_open$; alarm colour if NOT $lock$
rectangle at (0,0)-(31,31): invisible if NOT $open$
*)

(* Visualisation zLibrary/VisuObjects/INFO_TREE
1 elements of other kinds (tables, trends, ...) not read
*)

(* Visualisation 00_MainMenu(Tree)/M0000_MAIN
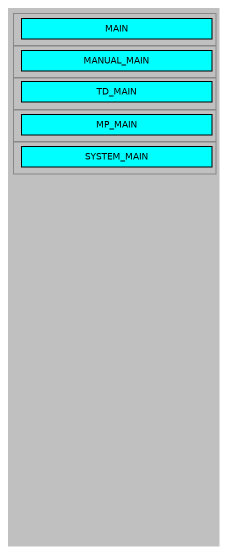
rectangle at (0,0)-(211,538): invisible if TRUE
embedded screen at (5,5)-(208,38): VISUBUTTON_TREE
embedded screen at (5,37)-(208,70): VISUBUTTON_TREE
embedded screen at (5,69)-(208,102): VISUBUTTON_TREE
embedded screen at (5,101)-(208,134): VISUBUTTON_TREE
embedded screen at (5,133)-(208,166): VISUBUTTON_TREE
rectangle at (13,10)-(204,31): text "MAIN"; invisible if TRUE
rectangle at (13,42)-(204,63): text "MANUAL_MAIN"; invisible if TRUE
rectangle at (13,73)-(204,94): text "TD_MAIN"; invisible if TRUE
rectangle at (13,106)-(204,127): text "MP_MAIN"; invisible if TRUE
rectangle at (13,138)-(204,159): text "SYSTEM_MAIN"; invisible if TRUE
*)

(* Visualisation 00_MainMenu(Tree)/M0000_MANUAL
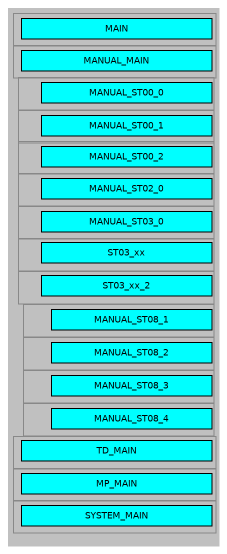
rectangle at (0,0)-(211,538): invisible if TRUE
embedded screen at (5,5)-(208,38): VISUBUTTON_TREE
embedded screen at (5,37)-(208,70): VISUBUTTON_TREE
embedded screen at (5,428)-(208,461): VISUBUTTON_TREE
embedded screen at (5,460)-(208,493): VISUBUTTON_TREE
embedded screen at (5,492)-(208,525): VISUBUTTON_TREE
rectangle at (13,10)-(204,31): text "MAIN"; invisible if TRUE
rectangle at (13,42)-(204,63): text "MANUAL_MAIN"; invisible if TRUE
rectangle at (13,432)-(204,453): text "TD_MAIN"; invisible if TRUE
rectangle at (13,465)-(204,486): text "MP_MAIN"; invisible if TRUE
rectangle at (13,497)-(204,518): text "SYSTEM_MAIN"; invisible if TRUE
embedded screen at (10,69)-(206,102): VISUBUTTON_TREE
rectangle at (33,74)-(204,95): text "MANUAL_ST00_0"; invisible if TRUE
embedded screen at (10,102)-(206,135): VISUBUTTON_TREE
rectangle at (33,107)-(204,128): text "MANUAL_ST00_1"; invisible if TRUE
embedded screen at (10,165)-(206,198): VISUBUTTON_TREE
rectangle at (33,170)-(204,191): text "MANUAL_ST02_0"; invisible if TRUE
embedded screen at (10,198)-(206,231): VISUBUTTON_TREE
rectangle at (33,203)-(204,224): text "MANUAL_ST03_0"; invisible if TRUE
embedded screen at (15,296)-(206,329): VISUBUTTON_TREE
rectangle at (43,301)-(204,322): text "MANUAL_ST08_1"; invisible if TRUE
embedded screen at (15,329)-(206,362): VISUBUTTON_TREE
rectangle at (43,334)-(204,355): text "MANUAL_ST08_2"; invisible if TRUE
embedded screen at (15,362)-(206,395): VISUBUTTON_TREE
rectangle at (43,367)-(204,388): text "MANUAL_ST08_3"; invisible if TRUE
embedded screen at (15,395)-(206,428): VISUBUTTON_TREE
rectangle at (43,400)-(204,421): text "MANUAL_ST08_4"; invisible if TRUE
embedded screen at (10,263)-(206,296): VISUBUTTON_TREE
embedded screen at (10,230)-(206,263): VISUBUTTON_TREE
rectangle at (33,267)-(204,288): text "ST03_xx_2"; invisible if TRUE
rectangle at (33,234)-(204,255): text "ST03_xx"; invisible if TRUE
embedded screen at (10,133)-(206,166): VISUBUTTON_TREE
rectangle at (33,138)-(204,159): text "MANUAL_ST00_2"; invisible if TRUE
*)

(* Visualisation 00_MainMenu(Tree)/M0002_MACHPARA
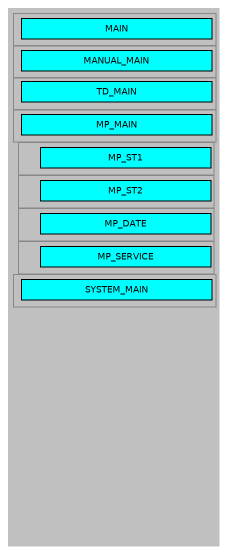
rectangle at (0,0)-(211,538): invisible if TRUE
embedded screen at (5,5)-(208,38): VISUBUTTON_TREE
embedded screen at (5,37)-(208,70): VISUBUTTON_TREE
embedded screen at (5,69)-(208,102): VISUBUTTON_TREE
embedded screen at (5,101)-(208,134): VISUBUTTON_TREE
embedded screen at (5,266)-(208,299): VISUBUTTON_TREE
rectangle at (13,10)-(204,31): text "MAIN"; invisible if TRUE
rectangle at (13,42)-(204,63): text "MANUAL_MAIN"; invisible if TRUE
rectangle at (13,73)-(204,94): text "TD_MAIN"; invisible if TRUE
rectangle at (13,106)-(204,127): text "MP_MAIN"; invisible if TRUE
rectangle at (13,271)-(204,292): text "SYSTEM_MAIN"; invisible if TRUE
embedded screen at (10,167)-(206,200): VISUBUTTON_TREE
rectangle at (32,172)-(203,193): text "MP_ST2"; invisible if TRUE
embedded screen at (10,200)-(206,233): VISUBUTTON_TREE
rectangle at (32,205)-(203,226): text "MP_DATE"; invisible if TRUE
embedded screen at (10,233)-(206,266): VISUBUTTON_TREE
rectangle at (32,238)-(203,259): text "MP_SERVICE"; invisible if TRUE
embedded screen at (10,134)-(206,167): VISUBUTTON_TREE
rectangle at (32,139)-(203,160): text "MP_ST1"; invisible if TRUE
*)

(* Visualisation 00_MainMenu(Tree)/M0003_SYSTEM
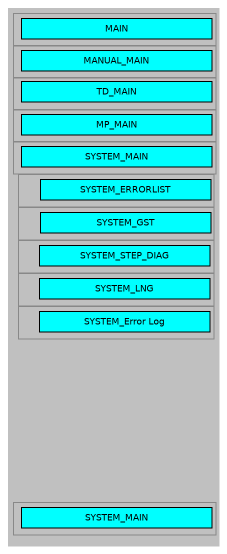
rectangle at (0,0)-(211,538): invisible if TRUE
embedded screen at (5,5)-(208,38): VISUBUTTON_TREE
embedded screen at (5,37)-(208,70): VISUBUTTON_TREE
embedded screen at (5,69)-(208,102): VISUBUTTON_TREE
embedded screen at (5,101)-(208,134): VISUBUTTON_TREE
embedded screen at (5,133)-(208,166): VISUBUTTON_TREE
rectangle at (13,10)-(204,31): text "MAIN"; invisible if TRUE
rectangle at (13,42)-(204,63): text "MANUAL_MAIN"; invisible if TRUE
rectangle at (13,73)-(204,94): text "TD_MAIN"; invisible if TRUE
rectangle at (13,106)-(204,127): text "MP_MAIN"; invisible if TRUE
rectangle at (13,138)-(204,159): text "SYSTEM_MAIN"; invisible if TRUE
embedded screen at (5,494)-(208,527): VISUBUTTON_TREE
rectangle at (13,499)-(204,520): text "SYSTEM_MAIN"; invisible if TRUE
embedded screen at (10,166)-(206,199): VISUBUTTON_TREE
rectangle at (32,171)-(203,192): text "SYSTEM_ERRORLIST"; invisible if TRUE
embedded screen at (10,199)-(206,232): VISUBUTTON_TREE
rectangle at (32,204)-(203,225): text "SYSTEM_GST"; invisible if TRUE
embedded screen at (10,232)-(206,265): VISUBUTTON_TREE
rectangle at (31,237)-(202,258): text "SYSTEM_STEP_DIAG"; invisible if TRUE
embedded screen at (10,265)-(206,298): VISUBUTTON_TREE
rectangle at (31,270)-(202,291): text "SYSTEM_LNG"; invisible if TRUE
embedded screen at (10,298)-(206,331): VISUBUTTON_TREE
rectangle at (31,303)-(202,324): text "SYSTEM_Error Log"; invisible if TRUE
*)

(* Visualisation 00_MainMenu(Tree)/M0003_TD
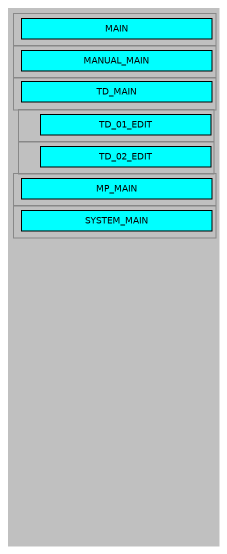
rectangle at (0,0)-(211,538): invisible if TRUE
embedded screen at (5,5)-(208,38): VISUBUTTON_TREE
embedded screen at (5,37)-(208,70): VISUBUTTON_TREE
embedded screen at (5,69)-(208,102): VISUBUTTON_TREE
embedded screen at (5,165)-(208,198): VISUBUTTON_TREE
embedded screen at (5,197)-(208,230): VISUBUTTON_TREE
rectangle at (13,10)-(204,31): text "MAIN"; invisible if TRUE
rectangle at (13,42)-(204,63): text "MANUAL_MAIN"; invisible if TRUE
rectangle at (13,73)-(204,94): text "TD_MAIN"; invisible if TRUE
rectangle at (13,170)-(204,191): text "MP_MAIN"; invisible if TRUE
rectangle at (13,202)-(204,223): text "SYSTEM_MAIN"; invisible if TRUE
embedded screen at (10,101)-(206,134): VISUBUTTON_TREE
rectangle at (32,106)-(203,127): text "TD_01_EDIT"; invisible if TRUE
embedded screen at (10,133)-(206,166): VISUBUTTON_TREE
rectangle at (32,138)-(203,159): text "TD_02_EDIT"; invisible if TRUE
*)

(* Visualisation 00_Main/MAIN
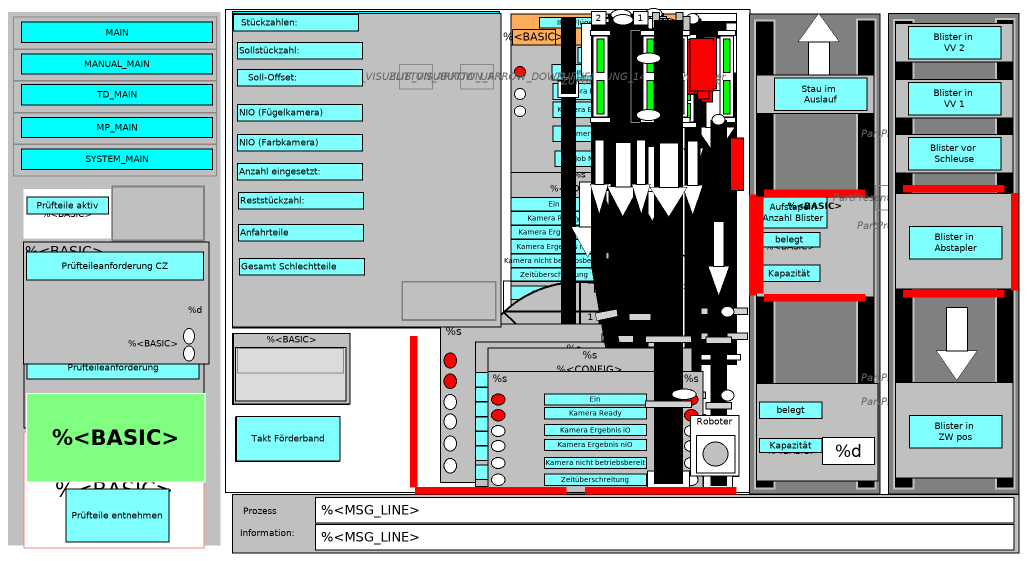
embedded screen at (220,111)-(745,597): ZUFUEHRUNG
rectangle at (227,597)-(1014,656): text "Prozess /  / Information:"
rectangle at (310,627)-(1009,653): text "%<MSG_LINE>"; shows ProcessMessage02; invisible if ProcessMessage02 = ''
rectangle at (310,600)-(1009,626): text "%<MSG_LINE>"; shows ProcessMessage01; invisible if ProcessMessage01=''
rectangle at (231,519)-(335,564): text "Takt Förderband"; invisible if TRUE
embedded screen at (744,116)-(875,597): WPC_Conveyor_Out
embedded screen at (898,492)-(923,517): PartPresentAndResult
embedded screen at (898,224)-(923,249): PartPresentAndResult
embedded screen at (3,115)-(215,648): M0000_Main
embedded screen at (898,468)-(923,493): PartPresentAndResult
embedded screen at (894,316)-(919,341): PartPresentAndResult
embedded screen at (870,288)-(895,313): PartPresentAndResult
embedded screen at (883,116)-(1014,597): WPC_CONVEYOR_IN
embedded screen at (18,283)-(204,651): PRUEFTEILENTNAHME
embedded screen at (227,116)-(496,430): TEILEZAEHLER
rectangle at (21,496)-(200,585): text "%<BASIC>"; shows 'Dummyprüfung aktiv'; invisible if NOT MP.ST02.DummyPruefung_93pol AND NOT DummyTest_160pol
rectangle at (228,436)-(345,507): text "%<BASIC>"; shows 'Föderband'; invisible if MP.ST03.SGM_3621
embedded screen at (230,450)-(341,504): ZLIB_OVERRIDE
rectangle at (685,518)-(734,579): text "Roboter"; opens MANUAL_ST03_0
embedded screen at (691,538)-(730,576): PARTRESULT
embedded screen at (410,590)-(561,597): DOOR_LOCK
embedded screen at (580,590)-(731,597): DOOR_LOCK
embedded screen at (405,439)-(412,590): DOOR_LOCK
1 elements of other kinds (tables, trends, ...) not read
*)

(* Visualisation 01_ManualMode/ST00/MANUAL_MAIN
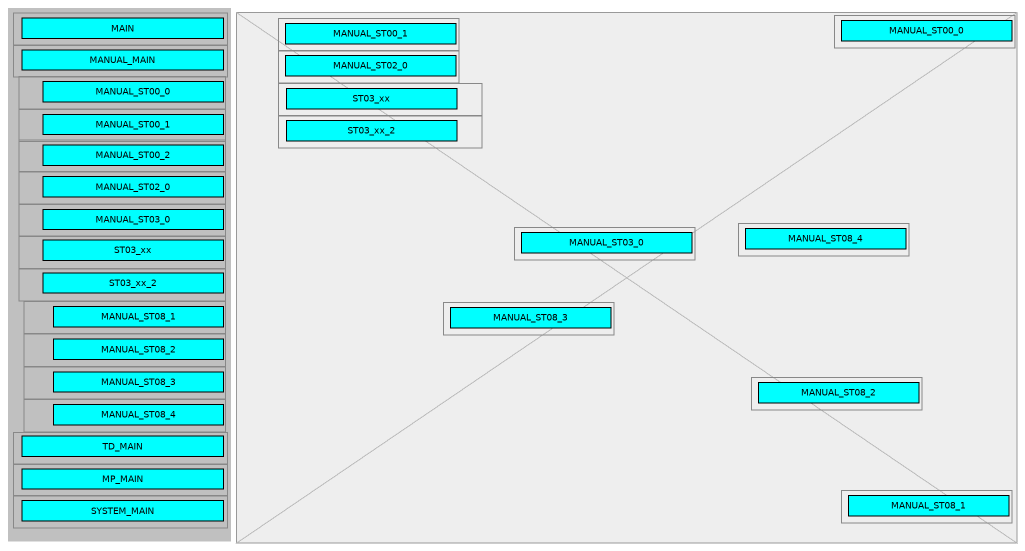
embedded screen at (3,115)-(226,648): M0000_Manual
bitmap at (231,119)-(1012,650): bmp\palettierer2.bmp
embedded screen at (273,125)-(454,158): VISUBUTTON_TREE
rectangle at (280,130)-(451,151): text "MANUAL_ST00_1"; invisible if TRUE
embedded screen at (273,157)-(454,190): VISUBUTTON_TREE
rectangle at (280,162)-(451,183): text "MANUAL_ST02_0"; invisible if TRUE
embedded screen at (509,334)-(690,367): VISUBUTTON_TREE
rectangle at (516,339)-(687,360): text "MANUAL_ST03_0"; invisible if TRUE
embedded screen at (836,597)-(1007,630): VISUBUTTON_TREE
rectangle at (843,602)-(1004,623): text "MANUAL_ST08_1"; invisible if TRUE
embedded screen at (746,484)-(917,517): VISUBUTTON_TREE
rectangle at (753,489)-(914,510): text "MANUAL_ST08_2"; invisible if TRUE
embedded screen at (438,409)-(609,442): VISUBUTTON_TREE
rectangle at (445,414)-(606,435): text "MANUAL_ST08_3"; invisible if TRUE
embedded screen at (733,330)-(904,363): VISUBUTTON_TREE
rectangle at (740,335)-(901,356): text "MANUAL_ST08_4"; invisible if TRUE
embedded screen at (829,122)-(1010,155): VISUBUTTON_TREE
rectangle at (836,127)-(1007,148): text "MANUAL_ST00_0"; invisible if TRUE
embedded screen at (273,190)-(477,223): VISUBUTTON_TREE
rectangle at (281,195)-(452,216): text "ST03_xx"; invisible if TRUE
embedded screen at (273,222)-(477,255): VISUBUTTON_TREE
rectangle at (281,227)-(452,248): text "ST03_xx_2"; invisible if TRUE
*)

(* Visualisation 01_ManualMode/ST00/MANUAL_ST00_0
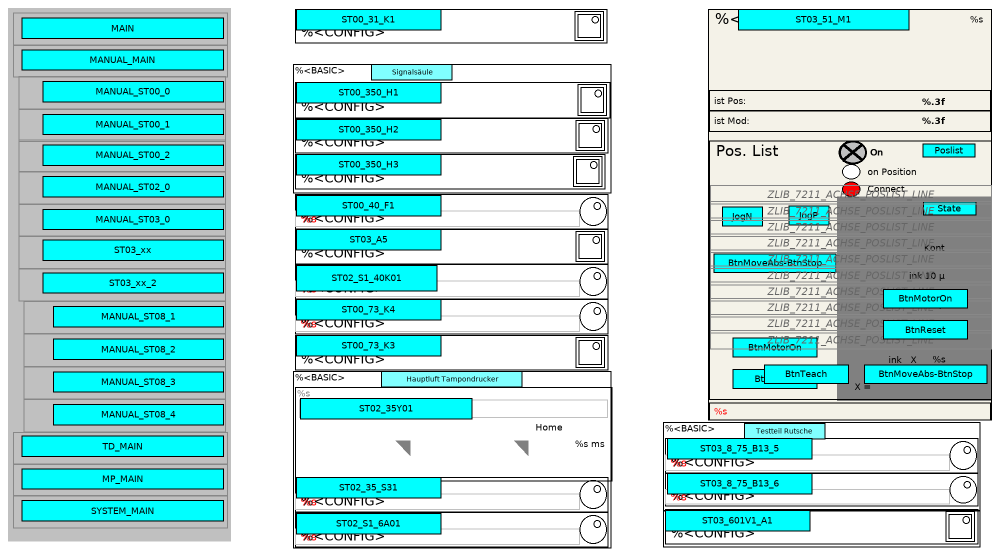
rectangle at (658,617)-(975,654): invisible if TD.TestpartBilister
embedded screen at (3,115)-(226,648): M0000_Manual
rectangle at (288,171)-(606,300): text "%<BASIC>"; shows 'Signalsäule'
embedded screen at (290,189)-(605,225): VDIGOUT_SMAL
embedded screen at (290,225)-(603,260): VDIGOUT_SMAL
embedded screen at (290,261)-(600,296): VDIGOUT_SMAL
embedded screen at (290,116)-(602,150): VDIGOUT_SMAL
embedded screen at (290,301)-(603,336): VDIGIN
embedded screen at (703,116)-(988,527): ZLIB_7211_Achse
embedded screen at (290,442)-(603,477): VDIGOUT_SMAL
rectangle at (288,478)-(606,655): text "%<BASIC>"; shows 'Tampondrucker'; invisible if gTypeCode<>4991 AND gTypeCode <>312
embedded screen at (290,584)-(603,619): VDIGIN
embedded screen at (290,494)-(607,588): ZLIB_VALVE_1_SENSORS
embedded screen at (290,619)-(603,654): VDIGIN
rectangle at (658,529)-(975,618): text "%<BASIC>"; shows 'Testteil Rutsche'; invisible if TD.TestpartBilister
embedded screen at (660,545)-(973,580): VDIGIN
embedded screen at (660,580)-(973,613): VDIGIN
embedded screen at (290,336)-(603,371): VDIGOUT_SMAL
rectangle at (739,530)-(820,546): text "Testteil Rutsche"; invisible if TRUE
rectangle at (366,171)-(447,187): text "Signalsäule"; invisible if TRUE
rectangle at (376,478)-(517,494): text "Hauptluft Tampondrucker"; invisible if TRUE
rectangle at (733,116)-(904,137): text "ST03_51_M1"; invisible if TRUE
embedded screen at (660,616)-(973,651): VDIGOUT_SMAL
rectangle at (295,505)-(467,526): text "ST02_35Y01"; invisible if TRUE
rectangle at (291,584)-(436,605): text "ST02_35_S31"; invisible if TRUE
rectangle at (291,620)-(436,641): text "ST02_S1_6A01"; invisible if TRUE
rectangle at (662,580)-(807,601): text "ST03_8_75_B13_6"; invisible if TRUE
rectangle at (662,545)-(807,566): text "ST03_8_75_B13_5"; invisible if TRUE
rectangle at (291,261)-(436,282): text "ST00_350_H3"; invisible if TRUE
rectangle at (291,442)-(436,463): text "ST00_73_K3"; invisible if TRUE
rectangle at (291,226)-(436,247): text "ST00_350_H2"; invisible if TRUE
rectangle at (291,189)-(436,210): text "ST00_350_H1"; invisible if TRUE
rectangle at (291,336)-(436,357): text "ST03_A5"; invisible if TRUE
rectangle at (660,617)-(805,638): text "ST03_601V1_A1"; invisible if TRUE
rectangle at (291,302)-(436,323): text "ST00_40_F1"; invisible if TRUE
rectangle at (291,116)-(436,137): text "ST00_31_K1"; invisible if TRUE
embedded screen at (290,406)-(603,441): VDIGIN
rectangle at (291,406)-(436,427): text "ST00_73_K4"; invisible if TRUE
embedded screen at (290,371)-(603,406): VDIGIN
rectangle at (291,372)-(432,398): text "ST02_S1_40K01"; invisible if TRUE
*)

(* Visualisation 01_ManualMode/ST00/MANUAL_ST00_1
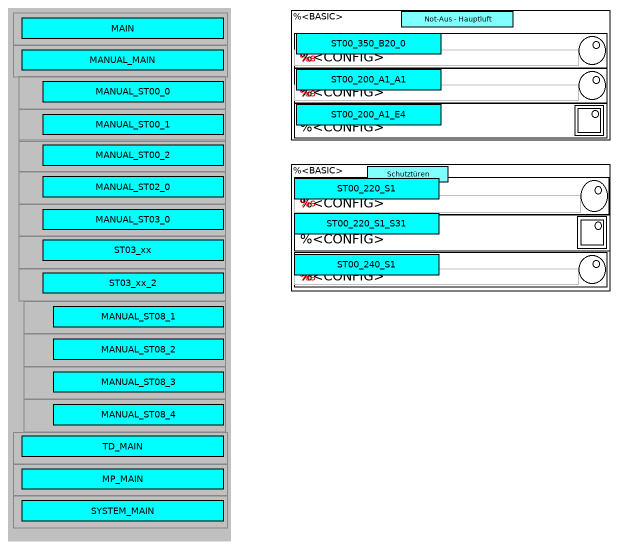
embedded screen at (3,115)-(226,648): M0000_Manual
rectangle at (286,271)-(605,398): text "%<BASIC>"; shows 'Schutztüren'
embedded screen at (289,321)-(605,358): VDIGOUT_SMAL
embedded screen at (289,284)-(604,322): VDIGIN
rectangle at (362,273)-(443,289): text "Schutztüren"; invisible if TRUE
rectangle at (289,320)-(434,341): text "ST00_220_S1_S31"; invisible if TRUE
rectangle at (289,285)-(434,306): text "ST00_220_S1"; invisible if TRUE
embedded screen at (289,359)-(602,394): VDIGIN
rectangle at (289,361)-(434,382): text "ST00_240_S1"; invisible if TRUE
rectangle at (286,117)-(605,247): text "%<BASIC>"; shows 'Not-Aus - Hauptluft'
embedded screen at (289,140)-(602,175): VDIGIN
embedded screen at (289,175)-(602,210): VDIGIN
embedded screen at (289,210)-(602,245): VDIGOUT_SMAL
rectangle at (396,118)-(508,134): text "Not-Aus - Hauptluft"; invisible if TRUE
rectangle at (291,140)-(436,161): text "ST00_350_B20_0"; invisible if TRUE
rectangle at (291,176)-(436,197): text "ST00_200_A1_A1"; invisible if TRUE
rectangle at (291,211)-(436,232): text "ST00_200_A1_E4"; invisible if TRUE
*)

(* Visualisation 01_ManualMode/ST00/MANUAL_ST00_2
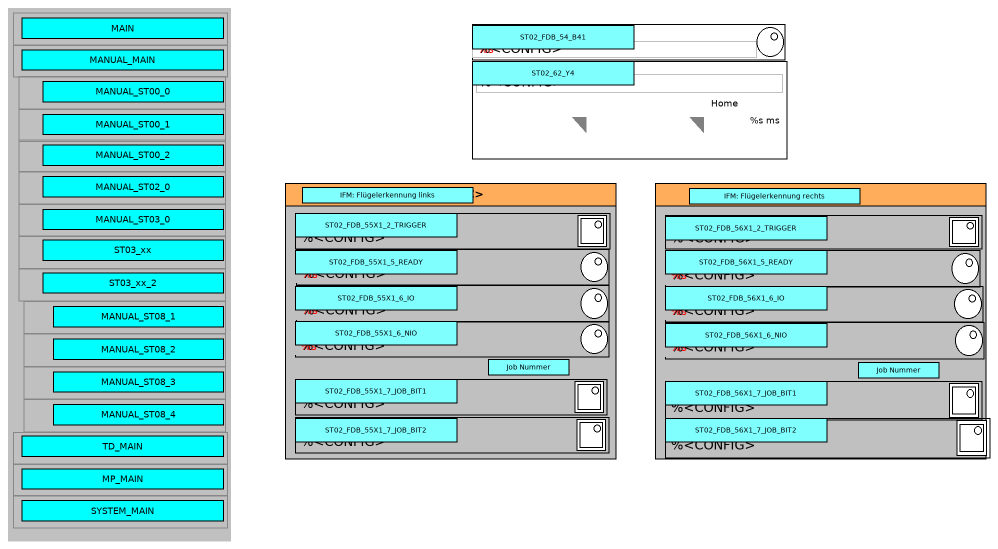
rectangle at (280,290)-(611,313): text "%<BASIC>"; shows 'IFM_Flügelerkennung_links'
rectangle at (650,290)-(981,313): text "%<BASIC>"; shows 'IFM_Flügelerkennung_rechts'
embedded screen at (3,115)-(226,648): M0000_Manual
embedded screen at (291,356)-(604,392): VDIGIN
embedded screen at (291,392)-(604,429): VDIGIN
embedded screen at (290,428)-(604,464): VDIGIN
embedded screen at (660,322)-(977,356): VDIGOUT_SMAL
embedded screen at (660,357)-(975,394): VDIGIN
embedded screen at (660,393)-(978,429): VDIGIN
embedded screen at (660,429)-(979,466): VDIGIN
embedded screen at (467,131)-(780,167): VDIGIN
embedded screen at (467,168)-(782,266): ZLIB_VALVE_1_SENSORS
embedded screen at (290,320)-(605,356): VDIGOUT_SMAL
embedded screen at (290,486)-(602,522): VDIGOUT_SMAL
embedded screen at (290,524)-(604,560): VDIGOUT_SMAL
embedded screen at (660,488)-(977,527): VDIGOUT_SMAL
embedded screen at (660,525)-(985,565): VDIGOUT_SMAL
rectangle at (297,294)-(468,310): text "IFM: Flügelerkennung links"; invisible if TRUE
rectangle at (684,295)-(855,311): text "IFM: Flügelerkennung rechts"; invisible if TRUE
rectangle at (481,464)-(562,483): text "%<BASIC>"; shows 'Job Nummer'
rectangle at (483,466)-(564,482): text "Job Nummer"; invisible if TRUE
rectangle at (851,467)-(932,486): text "%<BASIC>"; shows 'Job Nummer'
rectangle at (853,469)-(934,485): text "Job Nummer"; invisible if TRUE
rectangle at (290,486)-(452,510): text "ST02_FDB_55X1_7_JOB_BIT1"; invisible if TRUE
rectangle at (290,525)-(452,549): text "ST02_FDB_55X1_7_JOB_BIT2"; invisible if TRUE
rectangle at (290,428)-(452,452): text "ST02_FDB_55X1_6_NIO"; invisible if TRUE
rectangle at (290,393)-(452,417): text "ST02_FDB_55X1_6_IO"; invisible if TRUE
rectangle at (290,357)-(452,381): text "ST02_FDB_55X1_5_READY"; invisible if TRUE
rectangle at (290,320)-(452,344): text "ST02_FDB_55X1_2_TRIGGER"; invisible if TRUE
rectangle at (660,488)-(822,512): text "ST02_FDB_56X1_7_JOB_BIT1"; invisible if TRUE
rectangle at (660,525)-(822,549): text "ST02_FDB_56X1_7_JOB_BIT2"; invisible if TRUE
rectangle at (660,430)-(822,454): text "ST02_FDB_56X1_6_NIO"; invisible if TRUE
rectangle at (660,393)-(822,417): text "ST02_FDB_56X1_6_IO"; invisible if TRUE
rectangle at (660,357)-(822,381): text "ST02_FDB_56X1_5_READY"; invisible if TRUE
rectangle at (660,323)-(822,347): text "ST02_FDB_56X1_2_TRIGGER"; invisible if TRUE
rectangle at (467,132)-(629,156): text "ST02_FDB_54_B41"; invisible if TRUE
rectangle at (467,168)-(629,192): text "ST02_62_Y4"; invisible if TRUE
2 more shapes without text or variables
2 elements of other kinds (tables, trends, ...) not read
*)

(* Visualisation 01_ManualMode/ST02/MANUAL_ST02_0
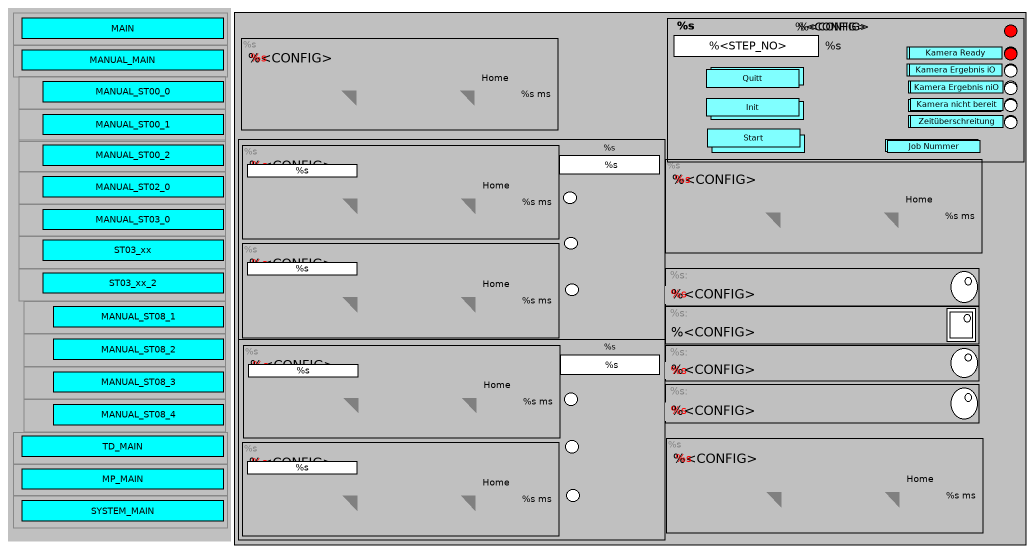
embedded screen at (3,115)-(226,648): M0000_Manual
rectangle at (233,246)-(660,447): alarm colour if ST02_62_Y6.SensorWorkIn[1].SensorSignal
rectangle at (233,446)-(660,647): alarm colour if ST02_62_Y6.SensorInitIn[1].SensorSignal
embedded screen at (660,413)-(974,451): VDIGOUT_SMAL
embedded screen at (236,145)-(553,237): ZLIB_VALVE_1_SENSORS
embedded screen at (660,452)-(974,488): VDIGIN
embedded screen at (237,350)-(554,445): ZLIB_VALVE_1_SENSORS
embedded screen at (237,252)-(554,346): ZLIB_VALVE_1_SENSORS
embedded screen at (237,549)-(554,643): ZLIB_VALVE_1_SENSORS
embedded screen at (238,452)-(555,545): ZLIB_VALVE_1_SENSORS
embedded screen at (552,249)-(657,422): ZLIB_Schwenkarm
embedded screen at (553,448)-(657,629): ZLIB_Schwenkarm
rectangle at (242,568)-(352,581): text "%s"; shows 'ST02_DT_61_B51'; alarm colour if ST02_DT_61_B51.ValveSensor
rectangle at (243,471)-(353,484): text "%s"; shows 'ST02_DT_61_B51'; alarm colour if ST02_DT_61_B51.ValveSensor
rectangle at (242,369)-(352,382): text "%s"; shows 'ST02_DT_61_B21'; alarm colour if ST02_DT_61_B21.ValveSensor
rectangle at (242,271)-(352,284): text "%s"; shows 'ST02_DT_61_B21'; alarm colour if ST02_DT_61_B21.ValveSensor
embedded screen at (660,375)-(974,413): VDIGIN
embedded screen at (660,491)-(974,530): VDIGIN
embedded screen at (661,545)-(978,640): ZLIB_VALVE_1_SENSORS
embedded screen at (660,266)-(977,360): ZLIB_VALVE_1_SENSORS
embedded screen at (662,125)-(1019,269): ZLIB_SENSOPART
embedded screen at (662,125)-(1019,269): ZLIB_SENSOPART_4
1 more shapes without text or variables
*)

(* Visualisation 01_ManualMode/ST03/MANUAL_ST03_0
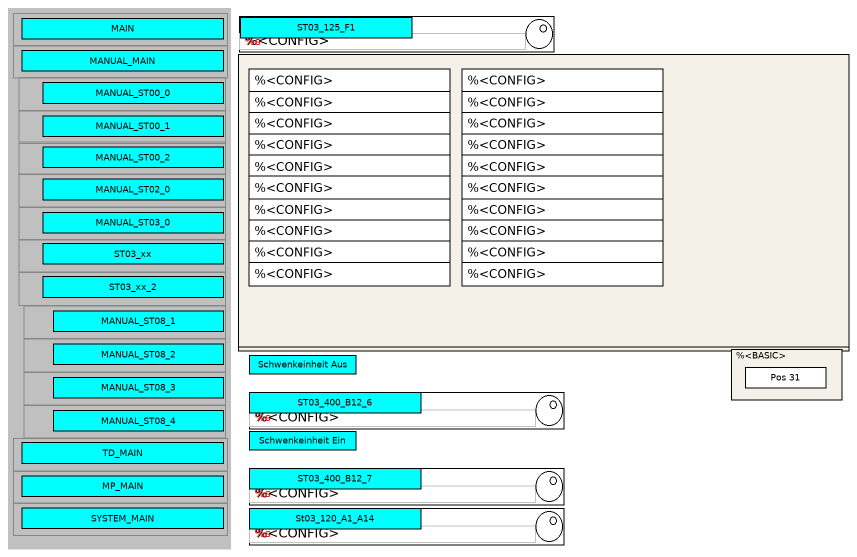
embedded screen at (3,115)-(226,656): M0000_Manual
embedded screen at (234,123)-(549,159): VDIGIN
embedded screen at (233,161)-(844,458): ZLIB_EPSON_ROBOT
embedded screen at (244,499)-(559,536): VDIGIN
embedded screen at (244,575)-(559,612): VDIGIN
embedded screen at (244,615)-(559,652): VDIGIN
rectangle at (244,538)-(351,557): text "Schwenkeinheit Ein"; invisible if TRUE
rectangle at (244,462)-(351,481): text "Schwenkeinheit Aus"; invisible if TRUE
rectangle at (235,124)-(407,145): text "ST03_125_F1"; invisible if TRUE
rectangle at (244,499)-(416,520): text "ST03_400_B12_6"; invisible if TRUE
rectangle at (244,575)-(416,596): text "ST03_400_B12_7"; invisible if TRUE
rectangle at (244,615)-(416,636): text "St03_120_A1_A14"; invisible if TRUE
group at (726,456)-(837,507)
  rectangle at (0,0)-(111,51): text "%<BASIC>"; shows 'Lageerkennung'
  rounded rectangle at (14,18)-(95,39): text "ERROR"
  rounded rectangle at (14,18)-(95,39): text "Pos 35"; invisible if ST03_Init_AbholPos.RoboPos31 AND ST03_Init_AbholPos.RoboPos35
  rounded rectangle at (14,18)-(95,39): text "Pos 31"; invisible if ST03_Init_AbholPos.RoboPos35; alarm colour if ST03_Init_AbholPos.RoboPos31
2 elements of other kinds (tables, trends, ...) not read
*)

(* Visualisation 01_ManualMode/ST03/MANUAL_ST03_1
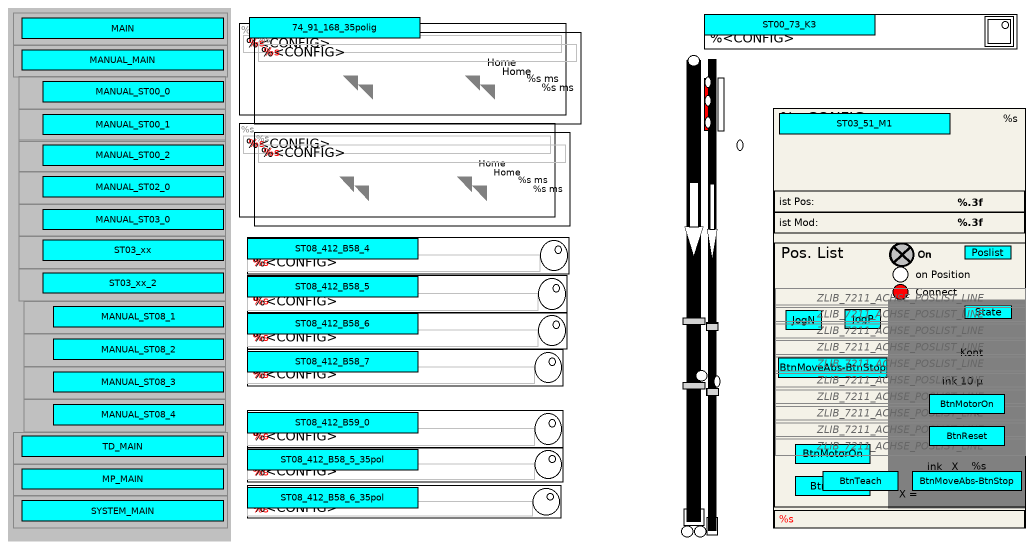
embedded screen at (3,115)-(226,648): M0000_Manual
embedded screen at (234,130)-(561,222): ZLIB_VALVE_1_SENSORS
embedded screen at (234,230)-(550,324): ZLIB_VALVE_1_SENSORS
embedded screen at (242,456)-(558,493): VDIGIN
embedded screen at (242,517)-(558,555): VDIGIN
embedded screen at (242,382)-(562,420): VDIGIN
embedded screen at (242,419)-(562,456): VDIGIN
embedded screen at (242,344)-(564,381): VDIGIN
embedded screen at (242,554)-(558,589): VDIGIN
embedded screen at (242,592)-(556,625): VDIGIN
embedded screen at (670,162)-(711,644): ZUFUEHRUNG_35POL
embedded screen at (697,166)-(738,642): ZUFUEHRUNG_74_91_168POL
embedded screen at (768,215)-(1022,635): ZLIB_7211_Achse
embedded screen at (249,139)-(576,231): ZLIB_VALVE_1_SENSORS
embedded screen at (249,239)-(565,333): ZLIB_VALVE_1_SENSORS
rectangle at (244,124)-(415,145): text "74_91_168_35polig"; invisible if TRUE
rectangle at (774,220)-(945,241): text "ST03_51_M1"; invisible if TRUE
rectangle at (242,345)-(413,366): text "ST08_412_B58_4"; invisible if TRUE
rectangle at (242,383)-(413,404): text "ST08_412_B58_5"; invisible if TRUE
rectangle at (242,420)-(413,441): text "ST08_412_B58_6"; invisible if TRUE
rectangle at (242,458)-(413,479): text "ST08_412_B58_7"; invisible if TRUE
rectangle at (242,519)-(413,540): text "ST08_412_B59_0"; invisible if TRUE
rectangle at (242,556)-(413,577): text "ST08_412_B58_5_35pol"; invisible if TRUE
rectangle at (242,594)-(413,615): text "ST08_412_B58_6_35pol"; invisible if TRUE
embedded screen at (699,121)-(1012,156): VDIGOUT_SMAL
rectangle at (699,121)-(870,142): text "ST00_73_K3"; invisible if TRUE
*)

(* Visualisation 01_ManualMode/ST03/MANUAL_ST03_10
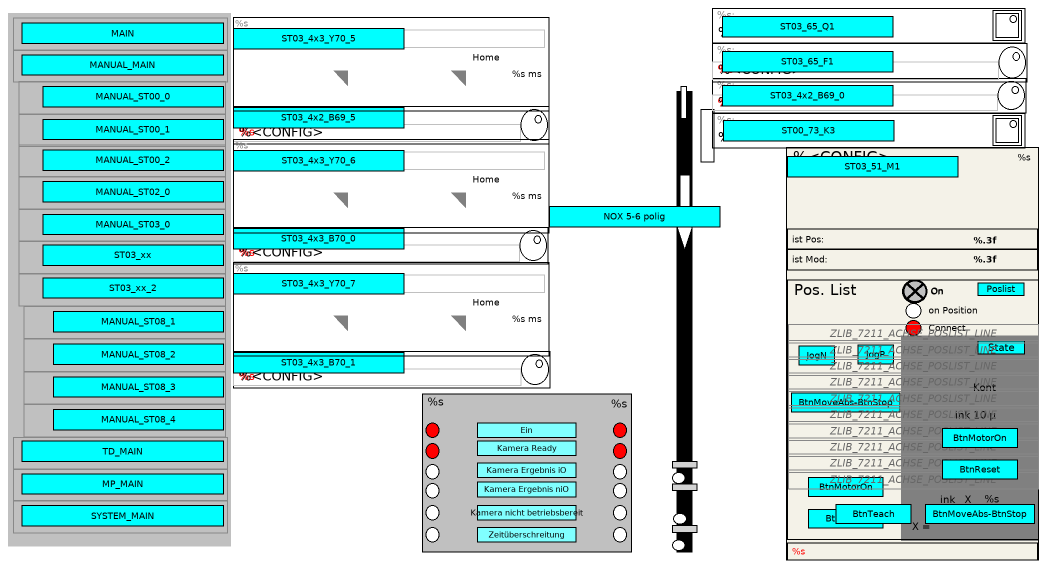
embedded screen at (3,115)-(226,648): M0000_Manual
embedded screen at (342,188)-(709,654): ZUFUEHRUNG_NOX_5_6POL
embedded screen at (228,453)-(545,490): VDIGIN
embedded screen at (707,180)-(1021,215): VDIGIN
embedded screen at (228,208)-(544,246): VDIGIN
embedded screen at (228,329)-(543,366): VDIGIN
embedded screen at (781,249)-(1035,662): ZLIB_7211_Achse
rectangle at (544,308)-(715,329): text "NOX 5-6 polig"; invisible if TRUE
rectangle at (717,187)-(888,208): text "ST03_4x2_B69_0"; invisible if TRUE
rectangle at (228,209)-(399,230): text "ST03_4x2_B69_5"; invisible if TRUE
rectangle at (228,454)-(399,475): text "ST03_4x3_B70_1"; invisible if TRUE
rectangle at (228,330)-(399,351): text "ST03_4x3_B70_0"; invisible if TRUE
rectangle at (782,258)-(953,279): text "ST03_51_M1"; invisible if TRUE
embedded screen at (228,119)-(544,213): ZLIB_VALVE_1_SENSORS
rectangle at (228,130)-(399,151): text "ST03_4x3_Y70_5"; invisible if TRUE
embedded screen at (228,241)-(544,335): ZLIB_VALVE_1_SENSORS
rectangle at (228,252)-(399,273): text "ST03_4x3_Y70_6"; invisible if TRUE
embedded screen at (228,364)-(544,458): ZLIB_VALVE_1_SENSORS
rectangle at (228,375)-(399,396): text "ST03_4x3_Y70_7"; invisible if TRUE
embedded screen at (707,110)-(1020,145): VDIGOUT_SMAL
rectangle at (717,118)-(888,139): text "ST03_65_Q1"; invisible if TRUE
embedded screen at (707,145)-(1022,184): VDIGIN
rectangle at (717,153)-(888,174): text "ST03_65_F1"; invisible if TRUE
embedded screen at (707,215)-(1020,250): VDIGOUT_SMAL
rectangle at (718,222)-(889,243): text "ST00_73_K3"; invisible if TRUE
*)

(* Visualisation 01_ManualMode/ST03/MANUAL_ST03_10_2
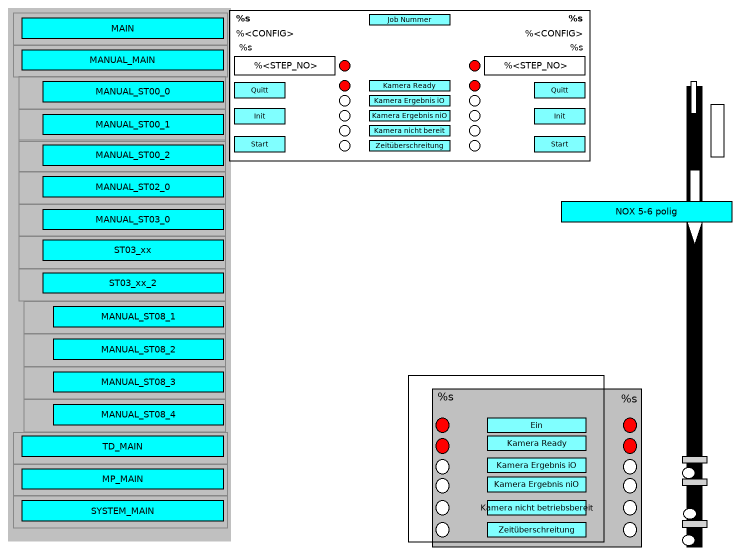
embedded screen at (3,115)-(226,648): M0000_Manual
embedded screen at (352,188)-(719,654): ZUFUEHRUNG_NOX_5_6POL
rectangle at (556,308)-(727,329): text "NOX 5-6 polig"; invisible if TRUE
embedded screen at (224,117)-(585,268): ZLIB_SENSOPART_4_2
1 more shapes without text or variables
*)

(* Visualisation 01_ManualMode/ST03/MANUAL_ST03_11
